INTERFACE ITF_MCMachineControl_HMI_Connector EXTENDS ITF_BaseTopElement_HMI_Connector

METHOD PUBLIC GetActiveMode : E_BaseMachineMode
VAR_INPUT
END_VAR
END_METHOD

METHOD PUBLIC GetActiveModeName : ST_BaseLabel
VAR_INPUT
END_VAR
END_METHOD

METHOD PUBLIC GetActiveState : E_BaseMachineState
VAR_INPUT
END_VAR
END_METHOD

METHOD PUBLIC GetActiveStateName : ST_BaseLabel
VAR_INPUT
END_VAR
END_METHOD

METHOD PUBLIC GetModeName : ST_BaseLabel
VAR_INPUT
	iNumber		: INT;
END_VAR
END_METHOD

METHOD PUBLIC GetStateName : ST_BaseLabel
VAR_INPUT
	iNumber		: INT;
END_VAR
END_METHOD

METHOD GetStateTimeForCurrentMode : LTIME
VAR_INPUT
	iNumber			: INT;
END_VAR
END_METHOD

METHOD GetStateTimeForMode : LTIME
VAR_INPUT
	iMode			: INT;
	iState			: INT;
END_VAR
END_METHOD

(*			
	RafalOS
	Rafał Osajda		24.11.2025		TC 4024.66
	Informacja czy dany stan jest aktywny w aktualnym trybie trybie
*)
METHOD PUBLIC IsStateActiveInCurrentMode : BOOL
VAR_INPUT
END_VAR
END_METHOD

METHOD PUBLIC SetCmdChangeState
VAR_INPUT
	eCmdNumber		: E_SaMCommandChangeState;
END_VAR
END_METHOD

END_INTERFACE

(* stored: Version 1.1.0.1
   Itf ITF_MCMachineControl_HMI_Connector: Id {d570e5d8-dcb3-079b-12de-407ccb79a8e5}
   Method GetActiveMode: Id {577b45bd-46f1-0f83-093b-77c467e398cb}
   Method GetActiveModeName: Id {4407dcff-23c5-0351-0a9c-547c33423be5}
   Method GetActiveState: Id {67cee8b6-905b-0059-03b5-535d5bad1116}
   Method GetActiveStateName: Id {0bb12475-6011-0270-1603-14ea9532c5e9}
   Method GetModeName: Id {ac65741e-56de-0aec-21f1-c2c7c554529c}
   Method GetStateName: Id {26719ab8-d41a-0159-05fa-021b5d6af891}
   Method GetStateTimeForCurrentMode: Id {89af58eb-efac-0122-3221-bddf27de8dd7}
   Method GetStateTimeForMode: Id {9d30221a-e7e7-09a7-2cea-e8b17dc27adc}
   Method IsStateActiveInCurrentMode: Id {a8b93514-5dce-08aa-0abb-b9e3c0d44ff0}
   Method SetCmdChangeState: Id {7447a1a1-d662-0680-3b3a-420ffd87d41f} *)
